FUNCTION_BLOCK PNEU_DRIVE
VAR_INPUT
END_VAR
VAR_OUTPUT
END_VAR
VAR
END_VAR

END_FUNCTION_BLOCK

(* stored: Version 1.1.0.1, ProductVersion 3.1.4022.18
   POU PNEU_DRIVE: Id {b535029c-b8c2-4b1f-9909-956f38e322b7}, SpecialFunc None *)
